KUKA KRL program: ros_rsi_110_fts.src

&ACCESS RVP
&PARAM TEMPLATE = C:\KRC\Roboter\Template\vorgabe
&PARAM EDITMASK = *
DEF ros_rsi_110_fts( )

; =============================================
;
; Software License Agreement (BSD License)
;
; Copyright (c) 2017 Norwegian University of Science and Technology
; All rights reserved.
;
; Redistribution and use in source and binary forms, with or without
; modification, are permitted provided that the following conditions
; are met:
;
;  * Redistributions of source code must retain the above copyright
;    notice, this list of conditions and the following disclaimer.
;  * Redistributions in binary form must reproduce the above
;    copyright notice, this list of conditions and the following
;    disclaimer in the documentation and/or other materials provided
;    with the distribution.
;  * Neither the name of the Norwegian University of Science and
;    Technology, nor the names of its contributors may be used to
;    endorse or promote products derived from this software without
;    specific prior written permission.
;
; THIS SOFTWARE IS PROVIDED BY THE COPYRIGHT HOLDERS AND CONTRIBUTORS
; "AS IS" AND ANY EXPRESS OR IMPLIED WARRANTIES, INCLUDING, BUT NOT
; LIMITED TO, THE IMPLIED WARRANTIES OF MERCHANTABILITY AND FITNESS
; FOR A PARTICULAR PURPOSE ARE DISCLAIMED. IN NO EVENT SHALL THE
; COPYRIGHT OWNER OR CONTRIBUTORS BE LIABLE FOR ANY DIRECT, INDIRECT,
; INCIDENTAL, SPECIAL, EXEMPLARY, OR CONSEQUENTIAL DAMAGES (INCLUDING,
; BUT NOT LIMITED TO, PROCUREMENT OF SUBSTITUTE GOODS OR SERVICES;
; LOSS OF USE, DATA, OR PROFITS; OR BUSINESS INTERRUPTION) HOWEVER
; CAUSED AND ON ANY THEORY OF LIABILITY, WHETHER IN CONTRACT, STRICT
; LIABILITY, OR TORT (INCLUDING NEGLIGENCE OR OTHERWISE) ARISING IN
; ANY WAY OUT OF THE USE OF THIS SOFTWARE, EVEN IF ADVISED OF THE
; POSSIBILITY OF SUCH DAMAGE.
;
; =============================================


; FOLD VAR DECLARATION
  CHAR configFileName[21]                    ;ST_ETHERNET object configuration file
  DECL RSIERR err                            ;Error value from RSI commands
  REAL lowerBound[12], upperBound[12]                ;Bounds for motion control

  INT i                                      ;Counter variable used in for-loops
  DECL AXIS HOME                             ; HOME position
  INT containerID, hEthernet, hAxis, hAnain[7], hDigin[16], hDigout[20], numAxes ;Container IDs
; ENDFOLD VAR DECLARATION

;FOLD INI
  ;FOLD BASISTECH INI
    GLOBAL INTERRUPT DECL 3 WHEN $STOPMESS==TRUE DO IR_STOPM ( )
    INTERRUPT ON 3
    BAS (#INITMOV,0 )
  ;ENDFOLD (BASISTECH INI)
  ;FOLD USER INI
    ;Make your modifications here

  ;ENDFOLD (USER INI)
;ENDFOLD (INI)

;FOLD Configuration
  numAxes = 6                                           ; Number of axes on robot
  HOME = {AXIS: A1 0, A2 -90, A3 90, A4 0, A5 90, A6 0} ; Start position
  configFileName[] = "ros_rsi_110_fts.xml"             ; Name of XML file. Should be in c:/krc/roboter/init

  ; Internal axes
  lowerBound[1] = -1000     ; lower limit A1 axis correction
  upperBound[1] =  1000     ; upper limit A1 axis correction
  lowerBound[2] = -1000     ; lower limit A2 axis correction
  upperBound[2] =  1000     ; upper limit A2 axis correction
  lowerBound[3] = -1000     ; lower limit A3 axis correction
  upperBound[3] =  1000     ; upper limit A3 axis correction
  lowerBound[4] = -1000     ; lower limit A4 axis correction
  upperBound[4] =  1000     ; upper limit A4 axis correction
  lowerBound[5] = -1000     ; lower limit A5 axis correction
  upperBound[5] =  1000     ; upper limit A5 axis correction
  lowerBound[6] = -1000     ; lower limit A6 axis correction
  upperBound[6] =  1000     ; upper limit A6 axis correction

  ; External axes
  lowerBound[7]  = -1000    ; lower limit E1 axis correction
  upperBound[7]  =  1000    ; upper limit E1 axis correction
  lowerBound[8]  = -1000    ; lower limit E2 axis correction
  upperBound[8]  =  1000    ; upper limit E2 axis correction
  lowerBound[9]  = -1000    ; lower limit E3 axis correction
  upperBound[9]  =  1000    ; upper limit E3 axis correction
  lowerBound[10] = -1000    ; lower limit E4 axis correction
  upperBound[10] =  1000    ; upper limit E4 axis correction
  lowerBound[11] = -1000    ; lower limit E5 axis correction
  upperBound[11] =  1000    ; upper limit E5 axis correction
  lowerBound[12] = -1000    ; lower limit E6 axis correction
  upperBound[12] =  1000    ; upper limit E6 axis correction



;ENDFOLD Configuration


; Move to start position
PTP $AXIS_ACT ; Be able to use PTP without all axes in HOME
;PTP HOME

; Create RSI Ethernet object
containerID = 0
err = ST_ETHERNET(hEthernet,containerID,configFileName[])
IF (err <> #RSIOK) THEN
  HALT
ENDIF

; Object for axis correction.
err = ST_AXISCORR(hAxis, containerID)
IF (err <> #RSIOK) THEN
  HALT
ENDIF

; Link axis correction objects from XML file
for i=1 TO numAxes
  err = ST_NEWLINK(hEthernet,i,hAxis,i)
  IF err<>#RSIOK  THEN
    HALT
  ENDIF
ENDFOR

; Set integration mode (0 absolute, 1 relative)
err = ST_SETPARAM(hAxis,1,0)
IF err<>#RSIOK THEN
  HALT
ENDIF

; Set lowerBound axis correction
for i=2 TO numAxes+1
  err = ST_SETPARAM(hAxis,i,lowerBound[i-1]);
  IF err<>#RSIOK THEN
    HALT
  ENDIF
ENDFOR

; Set upperBound axis correction
for i=14 TO numAxes+13
  err = ST_SETPARAM(hAxis,i,upperBound[i-13]);
  IF err<>#RSIOK THEN
    HALT
  ENDIF
ENDFOR

;Link Force Torque sensor without units
for i=1 TO 7
  err = ST_ANAIN(hAnain[i],0,i,0)
  err = ST_NEWLINK(hAnain[i],1,hEthernet,i)
ENDFOR

for i=1 TO 16
  err = ST_DIGIN(hDigin[i],0,i,0,0)
  err = ST_NEWLINK(hDigin[i],1,hEthernet,i+7)
ENDFOR

for i=1 TO 20
  err = ST_DIGOUT(hDigout[i],0,i,0,0)
  err = ST_NEWLINK(hDigout[i],1,hEthernet,i+23)
ENDFOR

; Start RSI execution
err = ST_ON()
IF (err <> #RSIOK) THEN
  HALT
ENDIF

; Runs untill RSI break
ST_SKIPSENS()

; Turn off RSI
err = ST_OFF()
IF (err <> #RSIOK) THEN
  HALT
ENDIF

; Go back to home position
; PTP HOME

END
